// TIA Portal V18 export
TYPE "quad_cnst_array"
// stored: IsFailsafeCompliant false
   STRUCT
      element : Array[0..3, 0..2] of Real;
   END_STRUCT;
   // element[0,0] := 0.00415;   // a
   // element[0,1] := 0.452;   // b
   // element[0,2] := 330.0;   // c
   // element[1,0] := -8.44E-07;   // a
   // element[1,1] := 0.000463;   // b
   // element[1,2] := 0.791;   // c
   // element[2,0] := -9.35E-05;   // a
   // element[2,1] := 0.000775;   // b
   // element[2,2] := 6.34;   // c
   // element[3,0] := -9.04E-05;   // a
   // element[3,1] := 0.0284;   // b
   // element[3,2] := 1.09;   // c
END_TYPE
